FUNCTION_BLOCK FB_Machine EXTENDS FB_PackML_BaseModule
VAR
	VirtualMaster : FB_VM		:= (Name := 'Virtual Master');
	Unwind		  : FB_Unwind	:= (Name := 'Unwind');
	Draw		  : FB_DrawAxis := (Name := 'Draw');
END_VAR

METHOD PUBLIC CyclicLogic
IF NOT InitComplete THEN
	_InitComplete := Initialize();
	RETURN;
END_IF

SUPER^.CyclicLogic();
END_METHOD

// Automatically enables and disables HMI control based on the PackML mode
METHOD PROTECTED HMIPermissions

// This method is called cyclically by CyclicLogic()
AllowHMIControl(ThisModuleOnly := TRUE);
END_METHOD

METHOD PROTECTED Initialize : BOOL;
VAR
	i						 : UDINT;
	varInfo					 : __SYSTEM.VAR_INFO;
	AllSubUnitsInitialized	 : BOOL := TRUE;
	AllComponentsInitialized : BOOL := TRUE;
END_VAR
Initialize := FALSE;
CASE DescendantSequenceState OF
	0:
		//Register Submodules
		RegisterSubmodule(VirtualMaster);
		RegisterSubmodule(Unwind);
		RegisterSubmodule(Draw);
		_LogModeChanges			:= FALSE;
		_LogStateChanges		:= FALSE;
		DescendantSequenceState := DescendantSequenceState + 10;

	10:
		//Setup Custom modes here
		DescendantSequenceState := DescendantSequenceState + 10;

	20: (* Default recipe values parameters entered here *)
		Unwind.MasterAxisRef	REF= VirtualMaster.AxisRef;
		Draw.MasterAxisRef		REF= VirtualMaster.AxisRef;
		DescendantSequenceState := DescendantSequenceState + 10;

	30:
		(* Copy Mode names *)
		FOR i := 1 TO 10 DO
			ModeNames[i] := F_UnitModeToString(UDINT_TO_DINT(i));
		END_FOR

		DescendantSequenceState := DescendantSequenceState + 10;

	40:
		(* Initialize Recipes *)
		DescendantSequenceState := DescendantSequenceState + 10;

	50:
		DescendantSequenceState := DescendantSequenceState + 10;

	60:
		IF SUPER^.Initialize() THEN
			DescendantSequenceState := DescendantSequenceState + 10;
		END_IF

	70:
		Initialize := TRUE;
END_CASE
END_METHOD

END_FUNCTION_BLOCK

(* stored: Version 1.1.0.1, ProductVersion 3.1.4024.12
   POU FB_Machine: Id {97b13e0f-7ef6-40f4-849d-6d84ce81f8c2}, SpecialFunc None
   Method CyclicLogic: Id {ebaa3bcd-61fa-4a47-a483-8bcc7204493f}
   Method HMIPermissions: Id {02a84cbc-9044-46fc-82ea-ae0aee99ae0f}
   Method Initialize: Id {7539f10c-75c9-45c6-b67b-8bf6d3682a5e} *)
